(* PLC project equipment_library, Dassault Systèmes ControlBuild 2024x *)
(* stored: creationDateTime 2023-10-03T11:13:33-01:00 *)

PROGRAM actuators

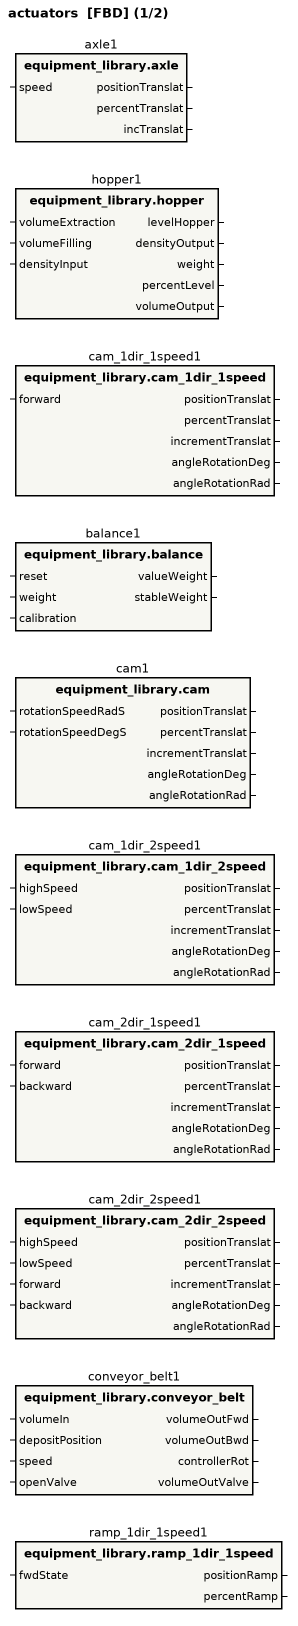
(* FBD diagram, written out as Structured Text *)
axle1();
hopper1();
cam_1dir_1speed1();
balance1();
cam1();
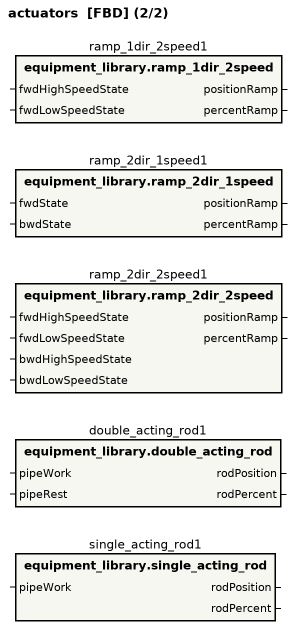
cam_1dir_2speed1();
cam_2dir_1speed1();
cam_2dir_2speed1();
conveyor_belt1();
ramp_1dir_1speed1();
ramp_1dir_2speed1();
ramp_2dir_1speed1();
ramp_2dir_2speed1();
double_acting_rod1();
single_acting_rod1();
END_PROGRAM

PROGRAM batch

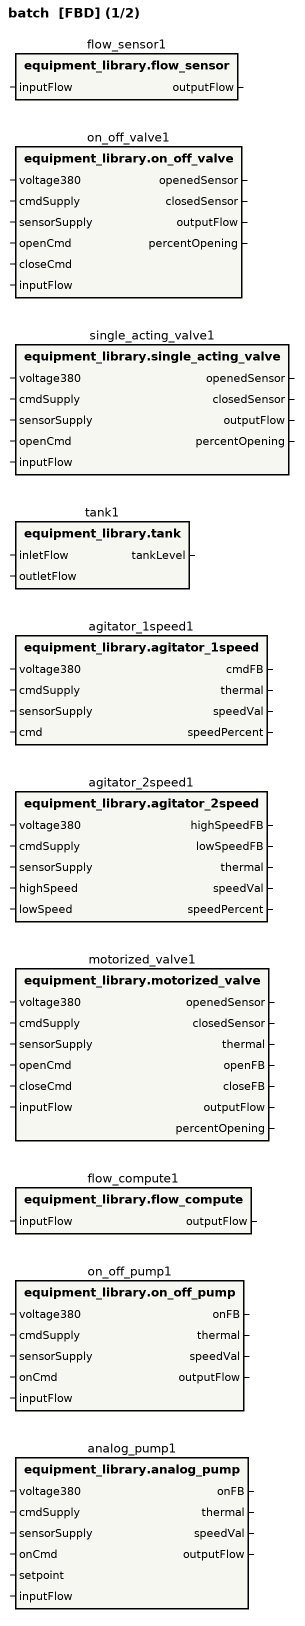
(* FBD diagram, written out as Structured Text *)
flow_sensor1();
on_off_valve1();
single_acting_valve1();
tank1();
agitator_1speed1();
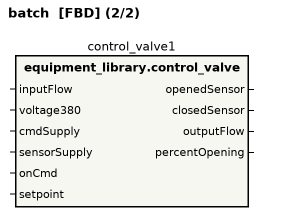
agitator_2speed1();
motorized_valve1();
flow_compute1();
on_off_pump1();
analog_pump1();
control_valve1();
END_PROGRAM

PROGRAM jacks

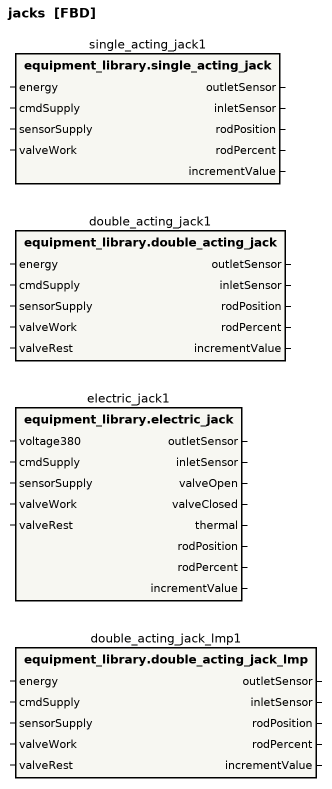
(* FBD diagram, written out as Structured Text *)
single_acting_jack1();
double_acting_jack1();
electric_jack1();
double_acting_jack_lmp1();
END_PROGRAM

PROGRAM motors

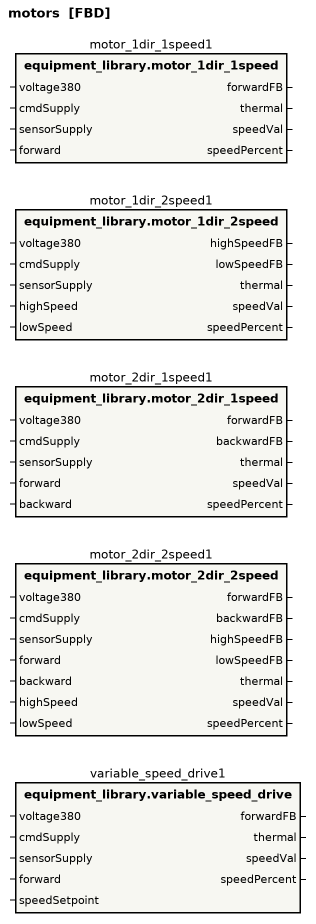
(* FBD diagram, written out as Structured Text *)
motor_1dir_1speed1();
motor_1dir_2speed1();
motor_2dir_1speed1();
motor_2dir_2speed1();
variable_speed_drive1();
END_PROGRAM

PROGRAM power

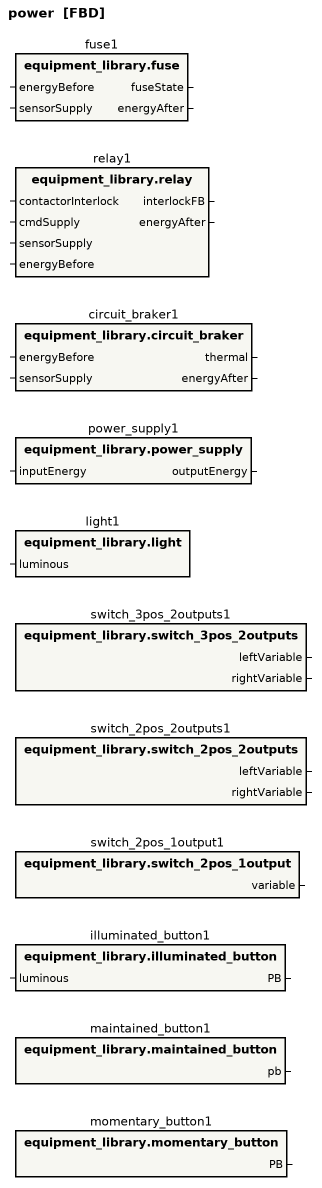
(* FBD diagram, written out as Structured Text *)
fuse1();
relay1();
circuit_braker1();
power_supply1();
light1();
switch_3pos_2outputs1();
switch_2pos_2outputs1();
switch_2pos_1output1();
illuminated_button1();
maintained_button1();
momentary_button1();
END_PROGRAM

PROGRAM preactuators

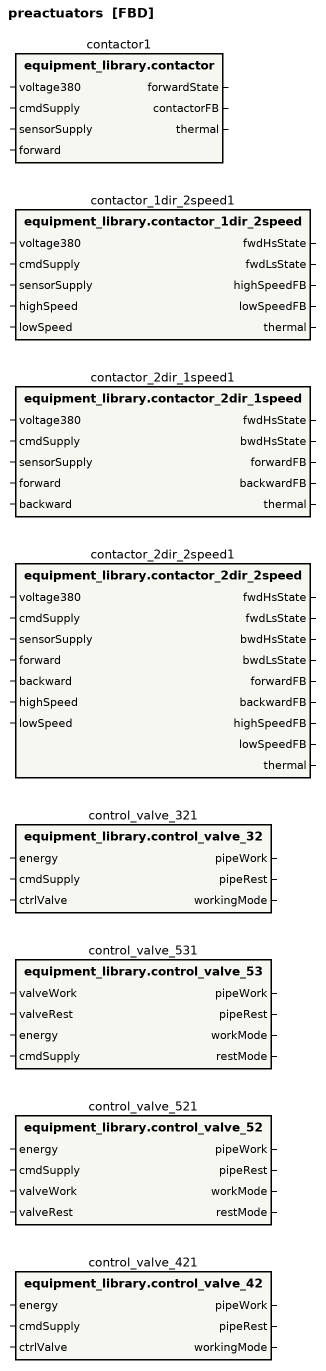
(* FBD diagram, written out as Structured Text *)
contactor1();
contactor_1dir_2speed1();
contactor_2dir_1speed1();
contactor_2dir_2speed1();
control_valve_321();
control_valve_531();
control_valve_521();
control_valve_421();
END_PROGRAM

PROGRAM sensors

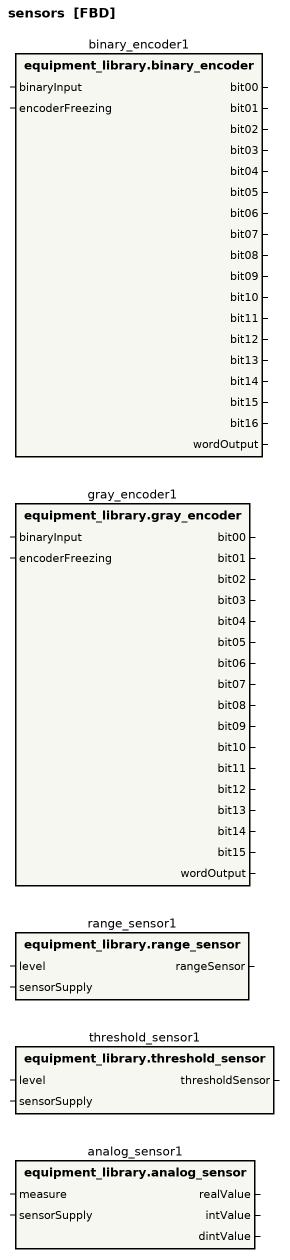
(* FBD diagram, written out as Structured Text *)
binary_encoder1();
gray_encoder1();
range_sensor1();
threshold_sensor1();
analog_sensor1();
END_PROGRAM

PROGRAM toolbox

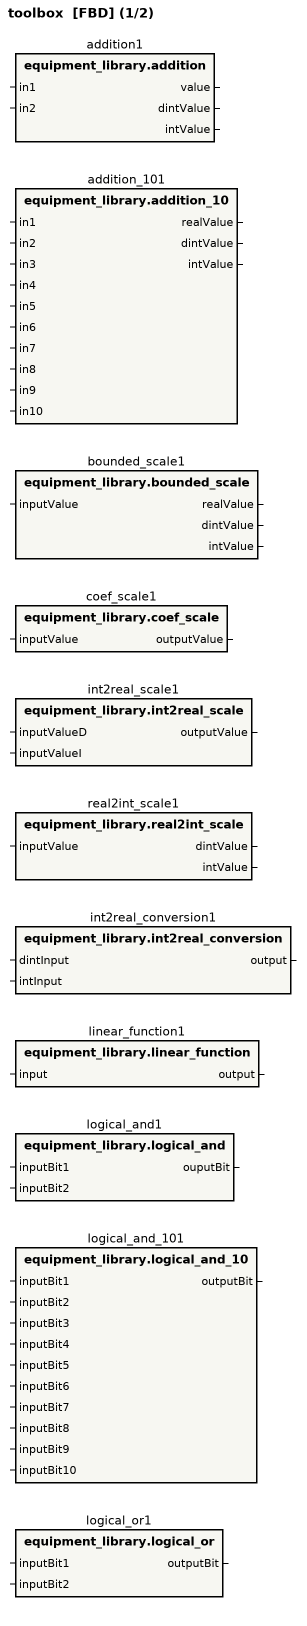
(* FBD diagram, written out as Structured Text *)
addition1();
addition_101();
bounded_scale1();
coef_scale1();
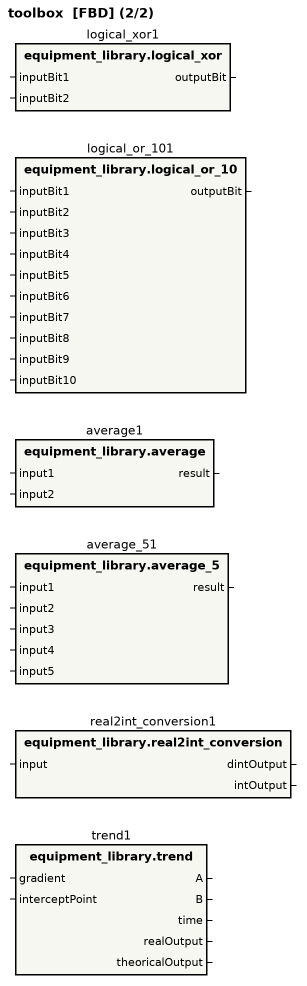
int2real_scale1();
real2int_scale1();
int2real_conversion1();
linear_function1();
logical_and1();
logical_and_101();
logical_or1();
logical_or_101();
logical_xor1();
average1();
average_51();
real2int_conversion1();
trend1();
END_PROGRAM

PROGRAM equipment_library.equipment_library

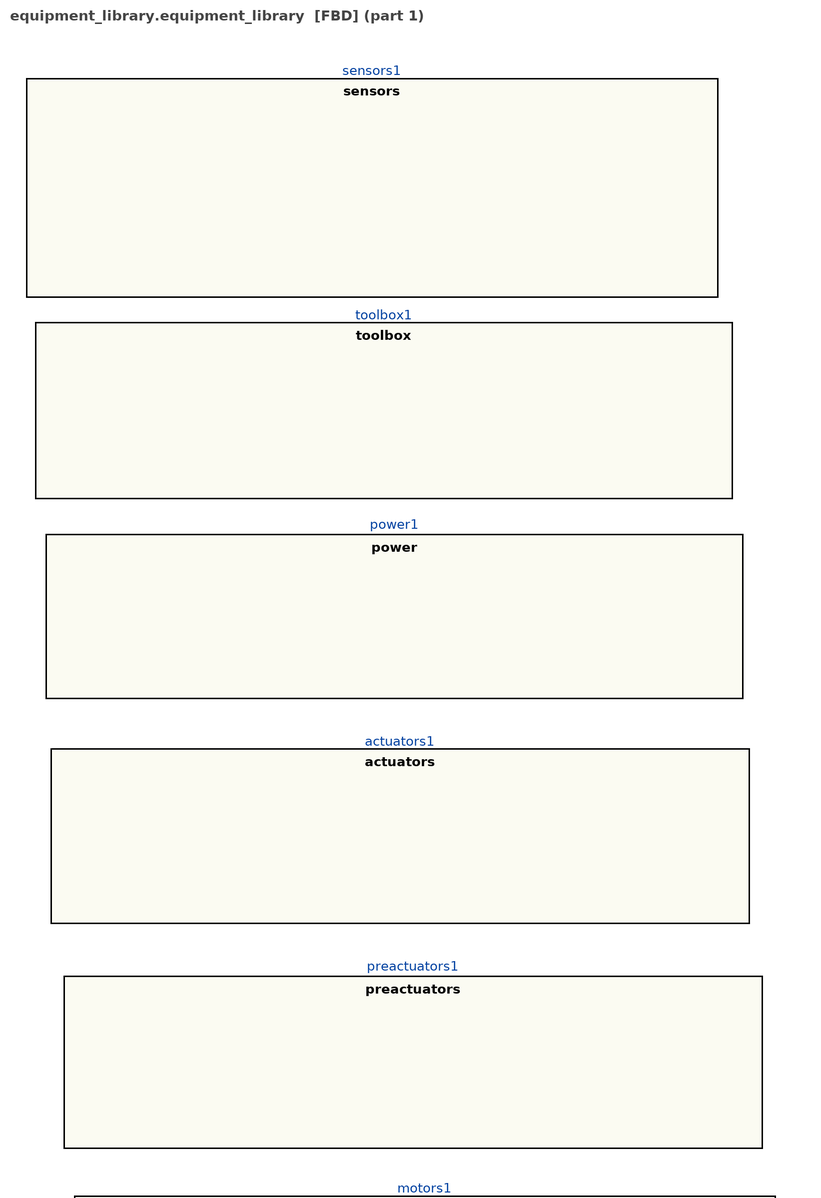
(* FBD diagram, written out as Structured Text *)
sensors1();
toolbox1();
power1();
actuators1();
preactuators1();
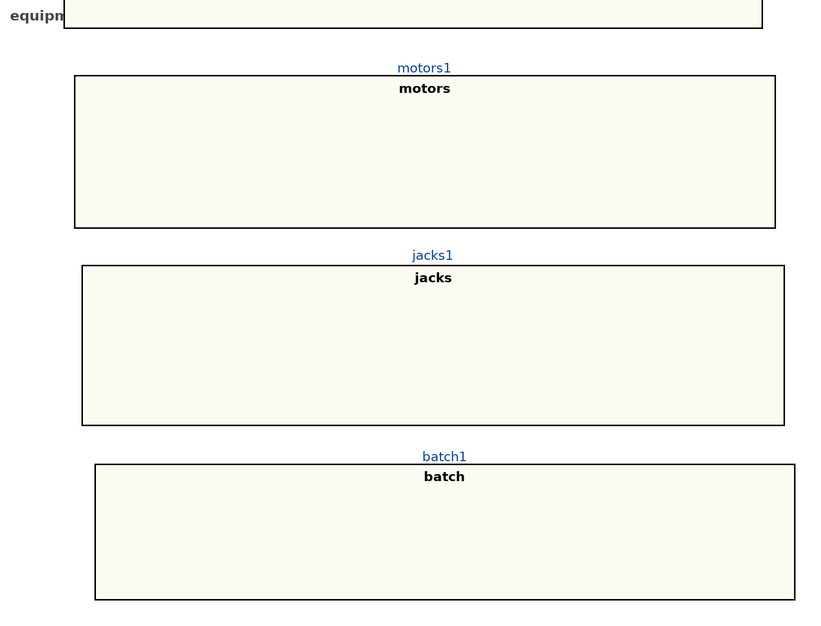
motors1();
jacks1();
batch1();
END_PROGRAM
